PROGRAM InvoerEnUitvoer
VAR

	StartUitvoer: BOOL;
	SensorUitvoer: Bool;
	MotorUitvoer: BOOL;
END_VAR

IF gvl.Power = TRUE THEN
		
	IF GVL.Initialisatie_voltooid = FALSE THEN
		Initialiseren();
	END_IF	
	
	IF GVL.Initialisatie_voltooid= TRUE AND GVL.startAanvoer =FALSE THEN 
			
			GVL.Status:= 'Voer de zaag lengte in';
			
	END_IF	

	IF GVL.ZaagLengte >= 0 AND GVL.StartAanvoer = TRUE THEN
		Simulatie_invoer();
		GVL.ZagenKlaar:=FALSE;
		sensorUitvoer := FALSE;
	END_IF
	
		
	IF GVL.ZaagLengte = GVL.HuidigePositieAanvoer AND motoruitvoer = FALSE AND gvl.ZagenKlaar = FALSE AND gvl.ZaagLengte >0 THEN
		gvl.AanvoerInPositie :=TRUE;
		GVL.StartAanvoer:=FALSE;
		GVL.Status:= 'Aanvoer in positie druk op: start zagen';
	END_IF
	
	
	IF GVL.ZagenKlaar THEN
		gvl.Status := 'Uitvoer actief';
		MotorUitvoer := TRUE;
	END_IF
	
	IF SensorUitvoer = TRUE AND gvl.ZagenKlaar THEN
		GVL.Status := 'Voer de zaaglengte in';
		MotorUitvoer := FALSE;
	END_IF
	
	
	
ELSE
	Gvl.MotorInvoer := FALSE;
	GVL.motoruitvoer := FALSE;
	
END_IF

END_PROGRAM

(* stored: Version 1.1.0.1, ProductVersion 3.1.4024.12
   POU InvoerEnUitvoer: Id {50253b7d-fc8b-4a12-9fbd-309ed75f9929}, SpecialFunc None *)
